// SIMATIC S7-200 project (STEP 7-Micro/WIN), CPU 222 REL 01.22

SYMBOL_TABLE USR1
FR1              I0.0     // RELE TERMICO
S1               I0.1     // PULSADOR PARO
S2               I0.2     // PULSADOR MARCHA
KM1              Q0.0     // CONTACTOR MARCHA
H1               Q0.1     // SEÑALIZACION MARCHA
H2               Q0.2     // SEÑALIZACION AVERIA
H3               Q0.3     // SEÑALIZACION PARARA
END_SYMBOL_TABLE

ORGANIZATION_BLOCK PRINCIPAL:OB1
TITLE=ARRANQUE DE UN MOTOR GUARDAMOTOR 
BEGIN
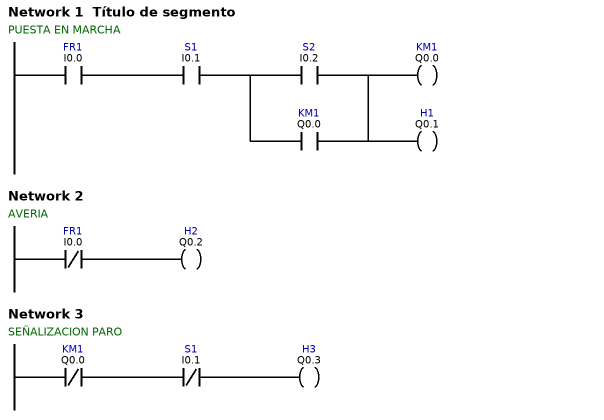
Network 1 // Título de segmento
// PUESTA EN MARCHA
LD     FR1:I0.0
A      S1:I0.1
LD     S2:I0.2
O      KM1:Q0.0
ALD
=      KM1:Q0.0
=      H1:Q0.1
Network 2
// AVERIA
LDN    FR1:I0.0
=      H2:Q0.2
Network 3
// SEÑALIZACION PARO
LDN    KM1:Q0.0
AN     S1:I0.1
=      H3:Q0.3
END_ORGANIZATION_BLOCK
